// Mitsubishi GX Developer project: Pumpim system PLC   PLC: FX1N

PROGRAM MAIN
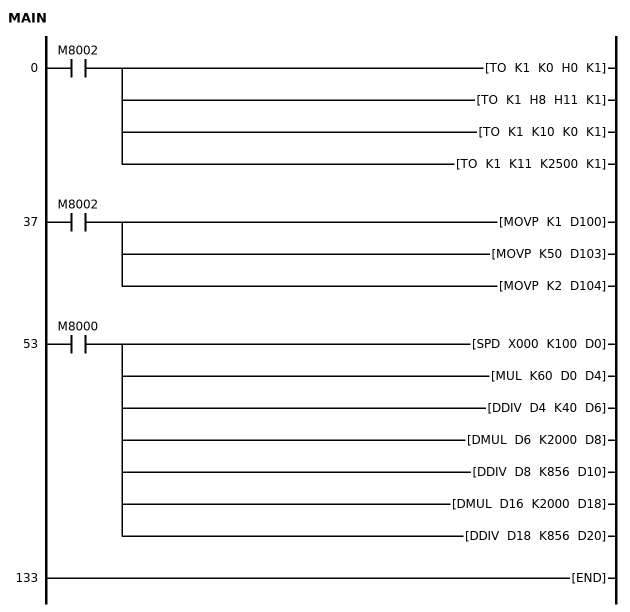
0     LD      M8002
      TO      K1 K0 H0 K1
        [note] DA Buffer #0
      TO      K1 H8 H11 K1
        [note] ENABLE OFFSET CH1&2
      TO      K1 K10 K0 K1
        [note] OFFSET VALUE CH1
      TO      K1 K11 K2500 K1
        [note] GAIN VALUE CH1
37    LD      M8002
      MOVP    K1 D100
        [note] PID PARAMTER SETING
      MOVP    K50 D103
      MOVP    K2 D104
53    LD      M8000
      SPD     X000 K100 D0
        [note] Speed Dectect
      MUL     K60 D0 D4
      DDIV    D4 K40 D6
      DMUL    D6 K2000 D8
      DDIV    D8 K856 D10
        [note] PV
      DMUL    D16 K2000 D18
      DDIV    D18 K856 D20
        [note] SV
133   END
END_PROGRAM
